Universal Robots PolyScope program: b_bot1.urp

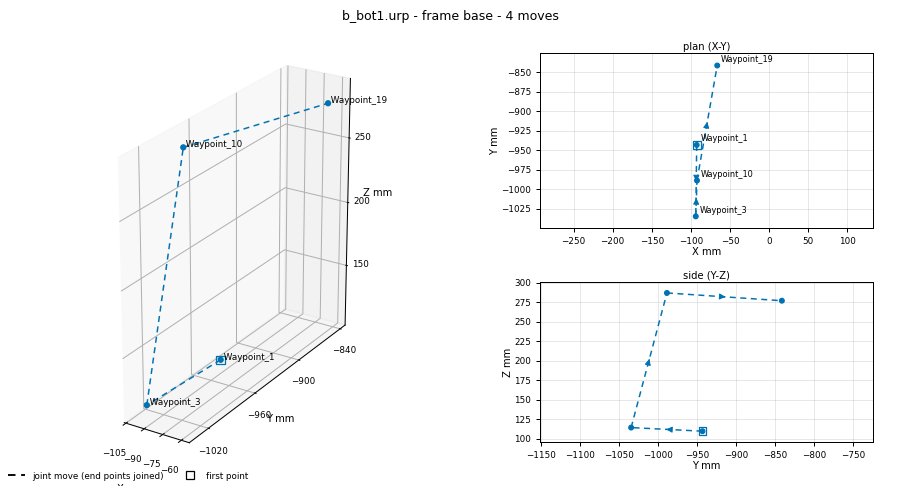
[picture p0: tool path of b_bot1.urp in frame base, 4 of 4 moves have a stored position in this frame; points joined in program order, loops and branches not executed]
Program b_bot1 (installation=default directory=/programs/Burkat_U_Plant createdIn=5.12.6.1102099 lastSavedIn=5.12.6.1102099 robotSerialNumber=20215500597)
Calibrated DH parameters: a=[0.000193, -0.066673, -0.391568, -0.000012, 0.00005, 0]; d=[0.162643, -472.05677, 465.132521, 7.058239, 0.099746, 0.099582]; alpha=[1.571116, 0.00089, 0.003862, 1.569269, -1.569248, 0]; deltaTheta=[0, -1.413394, 7.628392, 0.068187, 0, -0.000001]
Robot Program (runOnlyOnce=true)
  MoveJ speed 60 deg/s, acceleration 80 deg/s^2 (useActiveTCP=true) feature=Base
    Waypoint Waypoint_1: TCP in base x=-92.58 y=-943.208 z=109.706 mm, rx=1.5938 ry=0.0536 rz=-0.0777 rad; joints [70.625, -40.487, 74.961, -33.19, 71.628, -5.097] deg; TCP offset x=0 y=0 z=191.5 mm, rx=0 ry=0 rz=0 rad
  URCap Gripper (Robotiq_Grippers, Robotiq Inc.) dataModel(position=0.0, force=50.19607843137255, speed=26.19607843137255, positionInDouble=0.0, forceInDouble=50.19607843137255, speedInDouble=26.19607843137255, slaveIds=[9], blocking=true)
  MoveJ speed 60 deg/s, acceleration 80 deg/s^2 (useActiveTCP=true) feature=Base
    Waypoint Waypoint_3: TCP in base x=-93.764 y=-1034.535 z=114.342 mm, rx=1.6143 ry=0.0334 rz=-0.0505 rad; joints [72.827, -28.377, 48.902, -18.05, 73.535, -3.64] deg
  URCap Gripper (Robotiq_Grippers, Robotiq Inc.) dataModel(position=100.0, force=40.19607843137255, speed=26.19607843137255, positionInDouble=100.0, forceInDouble=40.19607843137255, speedInDouble=26.19607843137255, slaveIds=[9], blocking=true)
  MoveJ speed 40 deg/s, acceleration 80 deg/s^2 (useActiveTCP=true) feature=Base
    Waypoint Waypoint_10: TCP in base x=-92.228 y=-988.698 z=286.655 mm, rx=1.6465 ry=0.0332 rz=-0.0452 rad; joints [71.779, -43.319, 50.021, -2.274, 72.327, -4.08] deg
    Waypoint Waypoint_19: TCP in base x=-66.326 y=-841.615 z=276.687 mm, rx=1.6517 ry=-0.0259 rz=-0.093 rad; joints [71.48, -64.638, 86.648, -17.383, 75.945, -3.629] deg
